Yaskawa INFORM job: KRIS4(-224_-90)X2.JBI

/JOB
//NAME KRIS4(-224_-90)X2
//POS
///NPOS 317,317,317,14,0,0
///TOOL 0
///POSTYPE PULSE
///PULSE
C00000=126,-73357,-105376,-18827,72039,-77556
C00001=32651,40852,-26417,-15259,84054,10521
C00002=30282,121459,21655,-7232,82256,-84550
C00003=119678,189491,121384,-6609,55844,-83781
C00004=119958,189291,121101,-6814,55937,-83682
C00005=119958,189291,121101,-6814,104918,-83682
C00006=69507,150313,105301,-6814,83622,-83682
C00007=102374,11647,-10601,-6208,113224,-88139
C00008=49110,-96581,-90191,-6208,113224,-88139
C00009=-73090,-118428,-105692,-6208,113224,-88139
C00010=-121621,-118428,-105692,-6208,113224,-88139
C00011=72199,118597,79738,-6814,89727,-83682
C00012=-14837,117754,79738,-6814,55937,-83682
C00013=-44504,100666,44561,-7265,69044,-83737
C00014=-106120,216,-72664,-1265,72875,-87293
C00015=-133015,-103640,-65816,3996,83698,-82063
C00016=-132086,-97485,-64003,4135,58701,-800
C00017=-149065,-104779,-51399,-7594,43822,-5087
C00018=-150289,-91952,-48932,-6393,56924,-6348
C00019=-150393,-90903,-46944,-6418,56235,-6345
C00020=-150312,-91064,-47459,-6419,56476,-6331
C00021=-149346,-88536,-46306,-6590,57139,-6001
C00022=-150281,-91600,-48374,-6405,56765,-6336
C00023=-170298,-72142,-39060,-11518,57888,-13007
C00024=-170167,-71928,-38964,-11546,57956,-12963
C00025=-170167,-71173,-37488,-11610,57441,-12905
C00026=-170167,-71393,-37919,-11591,57591,-12921
C00027=-169145,-69698,-37147,-11804,58123,-12578
C00028=-170288,-72356,-39514,-11498,58052,-13018
C00029=-137447,-116054,-63762,-19682,56909,112
C00030=-108026,-108792,-54867,4103,57296,6110
C00031=-81416,-94598,-46445,196,58741,15925
C00032=-81757,-93684,-45677,246,58738,15800
C00033=-81757,-92858,-44382,247,58365,15799
C00034=-81757,-93619,-45575,246,58708,15800
C00035=-82768,-91970,-45027,393,59221,15429
C00036=-81930,-94457,-46518,272,58858,15736
C00037=-128580,-105651,-52299,6719,58617,-1362
C00038=-130033,-102824,-49114,6921,58227,-1914
C00039=-130033,-101283,-46878,6964,57648,-1951
C00040=-130033,-101721,-47515,6952,57813,-1940
C00041=-129738,-99854,-46987,6872,58421,-1793
C00042=-130056,-102692,-48758,6935,58079,-1930
C00043=-106734,-120076,-67764,3834,59373,6657
C00044=-106734,-120076,-67764,3834,76101,81400
C00045=-85493,-101158,-51309,10056,72841,87538
C00046=-85426,-99920,-49312,10091,72250,87511
C00047=-85426,-98477,-47146,10119,71667,87460
C00048=-85426,-98764,-47576,10113,71783,87469
C00049=-84550,-100156,-47986,10204,71224,87714
C00050=-85920,-99324,-49419,10033,72673,87380
C00051=-152431,-100504,-49770,2471,77391,65939
C00052=-152805,-100536,-48996,2423,76908,65809
C00053=-152805,-99353,-47240,2427,76436,65801
C00054=-152805,-99697,-47754,2425,76574,65803
C00055=-153892,-101565,-48290,2277,75972,65442
C00056=-152767,-100966,-49728,2425,77135,65826
C00057=-175766,-86349,-42944,-18121,68088,61743
C00058=-175951,-86348,-42668,-18137,67889,61707
C00059=-175951,-85124,-40623,-18213,67291,61803
C00060=-175951,-85392,-41070,-18196,67421,61782
C00061=-177474,-87024,-41664,-18224,66648,61355
C00062=-175558,-86298,-43164,-18103,68288,61786
C00063=-175558,-91829,-52585,-17786,71106,61349
C00064=-197698,-109667,-58160,-17366,61060,54816
C00065=-219000,-104945,-43712,-24315,53908,49637
C00066=-231055,-104193,-38505,-23952,48237,46148
C00067=-233659,-103437,-37306,-23712,47268,45306
C00068=-233659,-102004,-35373,-23879,46852,45418
C00069=-233659,-102412,-35924,-23830,46971,45386
C00070=-237043,-102549,-35954,-23321,46092,44173
C00071=-233629,-103481,-37368,-23709,47288,45313
C00072=-215461,-127400,-43893,-16870,58722,48272
C00073=-218544,-127186,-42626,-17459,57581,47480
C00074=-218544,-125569,-40789,-17514,57295,47527
C00075=-220330,-126171,-41362,-17770,57042,47002
C00076=-227145,-126469,-41362,-18757,55731,45038
C00077=-215464,-127169,-42828,-16963,58209,48354
C00078=-177088,-126078,-40365,-8704,67148,58850
C00079=-153631,-128510,-40310,-2158,67069,65285
C00080=-133342,-128267,-39542,4651,67425,70358
C00081=-133342,-124673,-35501,4672,66785,70333
C00082=-133342,-124996,-35867,4671,66843,70335
C00083=-136291,-126982,-35925,3818,65972,69519
C00084=-133342,-126415,-37468,4662,67098,70344
C00085=-196611,-116316,-69487,-12664,87450,51098
C00086=-193209,-126845,-128640,-12422,104242,50582
C00087=-154889,-136514,-128640,-12422,104242,50582
C00088=49700,-188138,-128640,-12422,104242,50582
C00089=95044,-166675,-127403,-9604,101606,54242
C00090=100905,-121879,-41170,-2953,61354,-13811
C00091=47156,-125376,-41742,-10980,55894,-30486
C00092=47156,-123817,-39951,-11019,55598,-30455
C00093=47156,-124234,-40431,-11009,55677,-30464
C00094=51773,-123508,-40415,-10441,56507,-29089
C00095=47156,-124816,-41100,-10994,55787,-30475
C00096=106085,-127336,-41103,-2720,58495,-12699
C00097=106085,-127336,-41103,-2720,58495,-12699
C00098=106085,-125446,-38966,-2726,58152,-12693
C00099=106085,-125807,-39375,-2725,58219,-12694
C00100=107264,-124702,-39383,-2517,58821,-12358
C00101=106085,-127485,-41271,-2717,58524,-12702
C00102=100408,-120926,-37847,15529,71533,-19798
C00103=97019,-119074,-33059,14623,70083,-20929
C00104=97019,-117387,-31072,14654,69737,-20973
C00105=97019,-117741,-31491,14648,69810,-20964
C00106=98849,-116641,-31480,15187,70099,-20422
C00107=96336,-121085,-34976,14390,70314,-21090
C00108=117002,-126078,-36297,14353,59540,-14518
C00109=129547,-123648,-35340,18268,59922,-11292
C00110=117730,-128646,-41030,15406,62632,-14363
C00111=118409,-131302,-43968,5246,61629,-11067
C00112=120969,-131398,-38796,6988,54321,-10972
C00113=120206,-131306,-38746,6863,54384,-11194
C00114=120401,-140874,-53529,6577,58526,-10873
C00115=92949,-132183,-43651,2261,56631,-10244
C00116=85861,-128380,-38765,-239,57883,-11923
C00117=85623,-128366,-38766,-283,57890,-11992
C00118=82836,-128240,-39082,-8880,55261,-11515
C00119=99554,-124935,-41395,-6066,59525,-6766
C00120=106086,-187684,-135216,-4534,68260,-4839
C00121=27739,-169745,-128413,-4049,68845,15832
C00122=-73947,-156826,-135344,-2505,79379,12508
C00123=-156474,-127565,-44757,-2910,70220,64434
C00124=-184477,-125463,-34959,-7013,67471,54171
C00125=-136126,-128460,-34213,11142,64994,67622
C00126=-154263,-130476,-42112,2655,69883,62096
C00127=-171605,-138664,-45039,-640,62750,56909
C00128=-183285,-124480,-40863,-3523,67329,53581
C00129=-201708,-124095,-40052,-8196,65992,48445
C00130=-164693,-130393,-40095,1325,64018,58749
C00131=-142889,-132361,-46546,6897,66121,64856
C00132=-228263,-110324,-43358,-23728,50162,46686
C00133=-235581,-106051,-39851,-22875,48410,44119
C00134=-236443,-96869,-37709,-21687,51363,43058
C00135=-226552,-115005,-54629,-22549,54767,46269
C00136=-203481,-118873,-57487,-18716,57337,53342
C00137=-209230,-112060,-51294,-18356,55868,51433
C00138=-214685,-102612,-48820,-17221,57967,49003
C00139=-205976,-112243,-55103,-18172,58669,52173
C00140=-201958,-123065,-58725,-3253,73839,54936
C00141=-198681,-127844,-56028,-6414,64844,57079
C00142=-178104,-136485,-56885,-3962,62059,63635
C00143=-171824,-140203,-61595,-3068,63271,65534
C00144=-141766,-147898,-61645,3344,56480,74079
C00145=-136469,-141007,-56961,2843,60494,76114
C00146=-120497,-136999,-55124,10696,63094,79702
C00147=-164064,-147455,-64185,5609,61717,65893
C00148=-164064,-147455,-64185,5609,61717,65893
C00149=-130860,-150279,-64151,-6173,30547,-11978
C00150=-181055,-130986,-61566,17152,51608,-35195
C00151=-181843,-125511,-58523,17019,52654,-35316
C00152=-83956,-132387,-59007,-5944,41709,3692
C00153=-101244,-134284,-58376,7865,38480,-5637
C00154=-129711,-151516,-73375,17379,42716,-18129
C00155=-134581,-137990,-74595,-25751,56070,1389
C00156=-110654,-139179,-74777,-26363,62443,9081
C00157=-115870,-127626,-66583,-26250,61756,7273
C00158=-184118,-104582,-60976,-13857,52675,-18268
C00159=-171621,-128341,-75090,-18129,51623,-12881
C00160=-119711,-181360,-121572,-24950,66300,4723
C00161=-89347,-163256,-129350,-23289,87878,11502
C00162=-119711,-181360,-135603,-24950,39029,4723
C00163=-119711,-181360,-135603,-24950,39029,4723
C00164=-67118,-136665,-130676,-31892,63753,-5674
C00165=-40548,-161800,-132385,-30407,51173,2851
C00166=-38594,-160347,-135413,-37506,33521,-5777
C00167=-38158,-160025,-136084,-39080,61805,-7690
C00168=-9060,-155984,-136090,-36075,61852,-27249
C00169=-9060,-155984,-136090,-36075,61852,-27249
C00170=35778,-73357,-105376,-18827,72039,-77556
C00171=35778,-73357,-105376,-18827,72039,-77556
C00172=121972,-60692,-66036,-23906,48760,-72917
C00173=121972,-63565,-66036,-13351,77444,-72917
C00174=114761,-44204,-50669,-11461,76826,-75375
C00175=114807,-42889,-47501,-11529,75582,-75243
C00176=114807,-42796,-46589,-11554,75077,-75195
C00177=114807,-42822,-46844,-11546,75217,-75208
C00178=114733,-44587,-47920,-11539,74967,-75210
C00179=114807,-42889,-47501,-11529,75582,-75243
C00180=106693,-40989,-47922,8584,79047,-76853
C00181=106712,-40732,-46990,8589,78608,-76878
C00182=106712,-40651,-45975,8604,78031,-76918
C00183=106712,-40674,-46241,8599,78181,-76908
C00184=106551,-42339,-47274,8643,77981,-76977
C00185=106693,-40989,-47922,8584,79047,-76853
C00186=119731,-42339,-42353,28777,73600,-71789
C00187=120080,-41537,-40336,28806,72749,-71870
C00188=120080,-41293,-39100,28897,72189,-72014
C00189=120080,-41335,-39305,28882,72281,-71990
C00190=120073,-43216,-40463,28920,72059,-72050
C00191=120080,-41537,-40336,28806,72749,-71870
C00192=101589,-42073,-44271,32201,81327,-76893
C00193=104782,-94542,-85411,8339,74693,-77861
C00194=98731,-154827,-131308,9878,72678,-80158
C00195=98731,-154827,-131308,9878,72678,-80158
C00196=98731,-154827,-131308,9878,72678,-80158
C00197=141095,-137804,-121947,-4358,90462,-65341
C00198=171917,-153174,-112370,11397,78411,-54227
C00199=199110,-110397,-63847,11158,69278,-59316
C00200=199661,-105459,-60576,13729,71348,-59282
C00201=199661,-104714,-59434,13753,71034,-59321
C00202=199661,-104881,-59692,13747,71104,-59313
C00203=201697,-105978,-60019,13785,70422,-58683
C00204=199661,-105459,-60576,13729,71348,-59282
C00205=123960,-138876,-68675,7989,69585,-84604
C00206=124072,-138705,-67366,8043,68864,-84619
C00207=124072,-137612,-66165,8049,68688,-84634
C00208=124072,-137824,-66399,8047,68723,-84632
C00209=124282,-139731,-66590,8126,67850,-84627
C00210=124072,-138655,-67314,8040,68857,-84622
C00211=114984,-139242,-68510,-12959,69151,-83072
C00212=114827,-138670,-67011,-13034,68516,-83052
C00213=114827,-136931,-65095,-13059,68238,-83020
C00214=114827,-137199,-65392,-13055,68282,-83025
C00215=114467,-139013,-65570,-13183,67430,-83044
C00216=114827,-138670,-67011,-13034,68516,-83052
C00217=133085,-142772,-85485,-9589,79895,-78262
C00218=119908,-107051,-70579,-11526,87272,-83253
C00219=119905,-107270,-70562,-11527,87152,-83243
C00220=119905,-106417,-69135,-11528,86722,-83203
C00221=119905,-106577,-69401,-11528,86804,-83211
C00222=119887,-108279,-69933,-11533,86265,-83166
C00223=119905,-107341,-70681,-11527,87191,-83247
C00224=147950,-101609,-70952,8097,88078,-75282
C00225=148936,-101577,-69519,8210,87121,-75014
C00226=148936,-100979,-68423,8210,86757,-75037
C00227=148936,-101159,-68752,8210,86867,-75032
C00228=149395,-102566,-69230,8263,86398,-74908
C00229=148936,-101830,-69986,8210,87277,-75005
C00230=165354,-89650,-65481,16319,85072,-70011
C00231=165779,-89873,-64407,16347,84242,-69973
C00232=165779,-89214,-62991,16359,83730,-70041
C00233=165779,-89312,-63202,16357,83805,-70031
C00234=166355,-90439,-63644,16386,83393,-69883
C00235=165632,-89756,-64683,16338,84492,-69992
C00236=143601,-106428,-78314,14904,88558,-77172
C00237=127839,-150907,-89343,18520,59767,-2936
C00238=132953,-138286,-79588,18019,59168,-1112
C00239=137115,-133470,-77672,17386,59565,529
C00240=137115,-131953,-75830,17447,59223,475
C00241=137115,-132842,-76915,17411,59423,507
C00242=136304,-129881,-76308,17304,60683,404
C00243=137115,-133253,-77414,17394,59515,521
C00244=181699,-110020,-71549,8619,60587,17610
C00245=181630,-109868,-71398,8637,60579,17583
C00246=181630,-109061,-70095,8670,60195,17555
C00247=181630,-109567,-70911,8650,60436,17574
C00248=179495,-107200,-70173,9064,61418,16842
C00249=181374,-109783,-71626,8682,60786,17501
C00250=138549,-156108,-92608,17680,56945,638
C00251=92857,-152389,-93170,-1138,51221,-11865
C00252=89241,-137374,-84375,-135,53495,-13313
C00253=89241,-137236,-84209,-135,53464,-13313
C00254=89241,-136248,-83020,-135,53240,-13313
C00255=89241,-136629,-83479,-135,53327,-13313
C00256=90422,-134246,-82978,-442,54247,-12852
C00257=88987,-137859,-84464,-69,53301,-13413
C00258=151501,-140988,-86034,-14129,58291,10466
C00259=150678,-138310,-84494,-13941,58574,10114
C00260=150678,-137164,-83136,-13977,58332,10146
C00261=150678,-137515,-83554,-13966,58407,10136
C00262=149186,-134345,-82896,-13563,59357,9449
C00263=151128,-139683,-85226,-14047,58399,10308
C00264=153806,-132474,-82078,-14195,60563,11039
C00265=88294,-133814,-82651,111,54267,-13684
C00266=119170,-146244,-89248,-14851,56054,5885
C00267=129919,-160370,-92966,12704,53201,-3154
C00268=134642,-143084,-81504,11683,54346,-1201
C00269=167270,-136117,-75530,1628,46891,11778
C00270=184998,-113755,-66262,10763,44700,16651
C00271=164928,-143381,-78407,9170,42235,9240
C00272=155273,-152427,-83467,13136,41921,4825
C00273=158141,-110882,-79211,11782,79402,-69500
C00274=156021,-110302,-75029,11867,77473,-70419
C00275=165528,-106206,-70771,11800,75600,-67301
C00276=175934,-96636,-67342,11366,76879,-63551
C00277=131080,-121620,-80305,3109,79327,-78003
C00278=138412,-119763,-75738,-25,77941,-75181
C00279=121865,-121897,-76297,-1096,77077,-80681
C00280=118816,-123903,-80121,-1281,78355,-81709
C00281=109990,-123163,-79929,-1817,78452,-84652
C00282=123486,-121654,-75594,-8156,77182,-79251
C00283=148715,-110583,-64793,-26650,87105,-69201
C00284=135969,-121502,-76764,-18008,81762,-74135
C00285=154667,-142334,-81197,-15526,77761,-67286
C00286=153773,-135579,-66423,-14508,74760,-67487
C00287=169136,-136018,-63121,-11093,74659,-62747
C00288=139166,-140952,-63595,-17941,67950,-71134
C00289=148278,-138995,-66659,-15795,72315,-68901
C00290=144415,-140880,-69264,8833,65243,-74412
C00291=148924,-141501,-67458,9395,63396,-73104
C00292=174434,-134936,-66673,11173,63406,-64720
C00293=167439,-135845,-70174,10586,65898,-66819
C00294=192902,-115042,-63146,20265,60680,-60371
C00295=201183,-110866,-58973,19481,58401,-57610
C00296=207998,-99743,-55745,17878,60466,-54609
C00297=170801,-131743,-76226,21430,65470,-67743
C00298=164740,-137810,-91614,20635,72894,-68588
C00299=164740,-137810,-91614,20635,72894,-68588
C00300=149447,-191890,-120181,21381,67024,-75156
C00301=149584,-192173,-120256,21405,66899,-75131
C00302=149584,-192173,-120256,21405,66899,-75131
C00303=114761,-44204,-50669,-11461,76826,-75375
C00304=117531,-39747,-45231,-12087,78952,-74614
C00305=125622,-38648,-38317,-31754,77240,-72218
C00306=114060,-50823,-52718,-11111,71580,-75110
C00307=124826,-51246,-53710,3634,72889,-70409
C00308=127047,-37417,-44991,3423,81297,-69380
C00309=134341,-35671,-43811,1894,81230,-66916
C00310=133954,-36259,-45628,1970,82055,-67034
C00311=135284,-28260,-32637,27547,76219,-65313
C00312=136540,-27437,-30649,27351,75093,-65095
C00313=137370,-25955,-24515,36210,70473,-65832
C00314=131832,-52683,-49405,33204,65462,-69826
C00315=109380,-75662,-60137,33198,63885,-64520
C00316=9054,-143647,-113334,-5954,77551,-79151
BC00000=192636,515545,1075136
BC00001=106856,514699,1075147
BC00002=45026,513209,1075136
BC00003=297205,515545,1075136
BC00004=388258,132939,1075136
BC00005=388258,132939,1075136
BC00006=266781,91691,1075136
BC00007=338196,12076,1075135
BC00008=385019,2960,1075135
BC00009=385019,2960,1075135
BC00010=335835,2960,1075135
BC00011=245343,24956,1075136
BC00012=171885,-116810,981693
BC00013=145068,-168564,1075136
BC00014=282408,-168564,1075136
BC00015=324871,12764,1075136
BC00016=324871,12764,1033476
BC00017=324871,12764,1033476
BC00018=324871,12764,1033476
BC00019=324871,12764,1033476
BC00020=324871,12764,1033476
BC00021=324871,12764,1033476
BC00022=324871,12764,1033476
BC00023=324871,12764,1033476
BC00024=324871,12764,1033476
BC00025=324871,12764,1033476
BC00026=324871,12764,1033476
BC00027=324871,12764,1033476
BC00028=324871,12764,1033476
BC00029=324871,12764,1033476
BC00030=324871,12764,1033476
BC00031=324871,12764,1033476
BC00032=324871,12764,1033476
BC00033=324871,12764,1033476
BC00034=324871,12764,1033476
BC00035=324871,12764,1033476
BC00036=324871,12764,1033476
BC00037=324871,12764,1033476
BC00038=324871,12764,1033476
BC00039=324871,12764,1033476
BC00040=324871,12764,1033476
BC00041=324871,12764,1033476
BC00042=324871,12764,1033476
BC00043=324871,12764,1033476
BC00044=324871,42664,1033476
BC00045=324871,42664,1033476
BC00046=324871,42664,1033476
BC00047=324871,42664,1033476
BC00048=324871,42664,1033476
BC00049=324871,42664,1033476
BC00050=324871,42664,1033476
BC00051=324871,42664,1033476
BC00052=324871,42664,1033476
BC00053=324871,42664,1033476
BC00054=324871,42664,1033476
BC00055=324871,42664,1033476
BC00056=324871,42664,1033476
BC00057=324871,42664,1033476
BC00058=324871,42664,1033476
BC00059=324871,42664,1033476
BC00060=324871,42664,1033476
BC00061=324871,42664,1033476
BC00062=324871,42664,1033476
BC00063=324871,42664,1033476
BC00064=324871,42664,1033476
BC00065=324871,70402,1033476
BC00066=324871,70402,1033476
BC00067=324871,70402,1033476
BC00068=324871,70402,1033476
BC00069=324871,70402,1033476
BC00070=324871,70402,1033476
BC00071=324871,70402,1033476
BC00072=324871,70402,1033476
BC00073=324871,70402,1033476
BC00074=324871,70402,1033476
BC00075=324871,70402,1033476
BC00076=324871,70402,1033476
BC00077=324871,70402,1033476
BC00078=346902,67759,1033476
BC00079=365604,67759,1033476
BC00080=358835,67759,1033476
BC00081=358835,67759,1033476
BC00082=358835,67759,1033476
BC00083=358835,67759,1033476
BC00084=358835,67759,1033476
BC00085=338593,67759,1033476
BC00086=365604,66159,1034603
BC00087=365604,17709,1034603
BC00088=365604,1629,1034603
BC00089=299593,3037,1034603
BC00090=314294,3037,1034603
BC00091=350319,4086,1007387
BC00092=350319,4086,1007387
BC00093=350319,4086,1007387
BC00094=350319,4086,1007387
BC00095=350319,4086,1007387
BC00096=302029,3926,1031408
BC00097=301345,10358,1012837
BC00098=301345,10358,1012837
BC00099=301345,10358,1012837
BC00100=301345,10358,1012837
BC00101=301345,10358,1012837
BC00102=302371,1302,1012837
BC00103=302371,1302,1012837
BC00104=302371,1302,1012837
BC00105=302371,1302,1012837
BC00106=302371,1302,1012837
BC00107=302371,1302,1012837
BC00108=302371,1302,1012837
BC00109=292881,1302,1012837
BC00110=310946,1302,1012837
BC00111=309160,1302,1012837
BC00112=309160,1302,1012837
BC00113=322422,1302,1012837
BC00114=322422,1302,1012837
BC00115=365717,2550,1012837
BC00116=365717,2550,1012837
BC00117=365717,2550,1012837
BC00118=365717,2550,1012837
BC00119=344627,2742,1042919
BC00120=344627,2742,1042919
BC00121=350887,22143,1073092
BC00122=276696,2854,1073092
BC00123=365604,67759,1033476
BC00124=354680,71198,1033476
BC00125=354680,71198,1033476
BC00126=354680,71198,1033476
BC00127=289396,71198,1033476
BC00128=299083,59780,1033476
BC00129=299083,59780,1033476
BC00130=299083,59780,1033476
BC00131=299083,59780,1033476
BC00132=323021,69640,1018791
BC00133=323021,69640,1018791
BC00134=323021,69640,1018791
BC00135=323021,69640,1018791
BC00136=323021,86344,1018791
BC00137=323020,86342,1018791
BC00138=323021,86344,1018791
BC00139=323021,86344,1018791
BC00140=323021,86344,1018791
BC00141=323021,86344,1018791
BC00142=323021,86344,1018791
BC00143=323021,86344,1018791
BC00144=359311,86344,1018791
BC00145=359311,86344,1018791
BC00146=359311,86344,1018791
BC00147=359311,86344,1018791
BC00148=320650,86344,1061699
BC00149=320650,38724,1061699
BC00150=348099,38724,988490
BC00151=348099,38724,988490
BC00152=348099,38724,988490
BC00153=348097,38726,988489
BC00154=348099,38724,988490
BC00155=348099,38724,988490
BC00156=317547,52292,963745
BC00157=317547,52292,963745
BC00158=317547,52292,963745
BC00159=317547,52292,963745
BC00160=317547,31600,963745
BC00161=278487,3584,1056780
BC00162=340345,-44387,1068891
BC00163=340345,-123490,1068891
BC00164=331767,-1766,1070081
BC00165=234698,5049,1063085
BC00166=254493,47555,1069374
BC00167=326806,106778,1070769
BC00168=344384,299723,1072198
BC00169=344384,446401,1072198
BC00170=295310,515545,1075136
BC00171=295310,513516,1075136
BC00172=295310,513263,813287
BC00173=335993,429318,731212
BC00174=335993,429318,731212
BC00175=335993,429318,731212
BC00176=335993,429318,731212
BC00177=335993,429318,731212
BC00178=335993,429318,731212
BC00179=335993,429318,731212
BC00180=292293,429318,731212
BC00181=292293,429318,731212
BC00182=292293,429318,731212
BC00183=292293,429318,731212
BC00184=292293,429318,731212
BC00185=292293,429318,731212
BC00186=292293,429318,731212
BC00187=292293,429318,731212
BC00188=292293,429318,731212
BC00189=292293,429318,731212
BC00190=292293,429318,731212
BC00191=292293,429318,731212
BC00192=292293,429318,731212
BC00193=292293,429318,731212
BC00194=292293,429318,979834
BC00195=314373,292172,979834
BC00196=314373,275872,695664
BC00197=349600,266255,695664
BC00198=349600,243768,695664
BC00199=318481,229664,891298
BC00200=318481,229664,891298
BC00201=318481,229664,891298
BC00202=318481,229664,891298
BC00203=318481,229664,891298
BC00204=318481,229664,891298
BC00205=318481,229664,891298
BC00206=318481,229664,891298
BC00207=318481,229664,891298
BC00208=318481,229664,891298
BC00209=318481,229664,891298
BC00210=318481,229664,891298
BC00211=347990,229664,891297
BC00212=347990,229664,891297
BC00213=347990,229664,891297
BC00214=347990,229664,891297
BC00215=347990,229664,891297
BC00216=347990,229664,891297
BC00217=347990,229664,891297
BC00218=347990,229664,891297
BC00219=347990,229664,891297
BC00220=347990,229664,891297
BC00221=347990,229664,891297
BC00222=347990,229664,891297
BC00223=347990,229664,891297
BC00224=347990,229664,891297
BC00225=347990,229664,891297
BC00226=347990,229664,891297
BC00227=347990,229664,891297
BC00228=347990,229664,891297
BC00229=347990,229664,891297
BC00230=317379,229664,891297
BC00231=317379,229664,891297
BC00232=317379,229664,891297
BC00233=317379,229664,891297
BC00234=317379,229664,891297
BC00235=317379,229664,891297
BC00236=317379,229664,891297
BC00237=317379,229664,891297
BC00238=317379,229664,891297
BC00239=317379,229664,891297
BC00240=317379,229664,891297
BC00241=317379,229664,891297
BC00242=317379,229664,891297
BC00243=317379,229664,891297
BC00244=317379,229664,891297
BC00245=317379,229664,891297
BC00246=317379,229664,891297
BC00247=317379,229664,891297
BC00248=317379,229664,891297
BC00249=317379,229664,891297
BC00250=317379,229664,891297
BC00251=339726,229664,891297
BC00252=339725,229663,891294
BC00253=339725,229663,891294
BC00254=339725,229663,891294
BC00255=339725,229663,891294
BC00256=339725,229663,891294
BC00257=339725,229663,891294
BC00258=339725,229663,891294
BC00259=339725,229663,891294
BC00260=339725,229663,891294
BC00261=339725,229663,891294
BC00262=339725,229663,891294
BC00263=339725,229663,891294
BC00264=339725,229663,891294
BC00265=339725,229663,891294
BC00266=339725,229663,891294
BC00267=310311,229663,891294
BC00268=310311,229663,891294
BC00269=310311,229663,891294
BC00270=310311,229663,891294
BC00271=310311,229663,891294
BC00272=310311,229663,891294
BC00273=310311,229663,891294
BC00274=310311,229663,891294
BC00275=310311,229663,891294
BC00276=310311,229663,891294
BC00277=310311,229663,891294
BC00278=310311,229663,891294
BC00279=310311,229663,891290
BC00280=310311,229663,891290
BC00281=351185,229663,891290
BC00282=351185,229663,891290
BC00283=351184,229663,891289
BC00284=351185,229663,891290
BC00285=351185,229663,891290
BC00286=351185,229663,891290
BC00287=351185,229663,891290
BC00288=351185,229663,891290
BC00289=351185,229663,891290
BC00290=335351,229663,891290
BC00291=335351,229663,891290
BC00292=335351,229663,891290
BC00293=335351,229663,891290
BC00294=335351,229663,891290
BC00295=335351,229663,891290
BC00296=335351,229663,891290
BC00297=335351,229663,891290
BC00298=335351,229663,891290
BC00299=352732,229663,1069777
BC00300=352732,229663,1069777
BC00301=352732,347909,1069777
BC00302=352732,347909,743295
BC00303=335993,429318,731212
BC00304=335994,429318,731211
BC00305=335994,429317,731208
BC00306=335994,429318,731211
BC00307=335994,429318,731211
BC00308=335994,429318,731211
BC00309=335994,429318,731211
BC00310=335994,429318,731211
BC00311=335994,429318,731211
BC00312=335994,429318,731211
BC00313=335994,429318,731211
BC00314=335994,429318,731211
BC00315=361465,487090,979283
BC00316=361465,516139,979283
EC00000=1986524,372644
EC00001=1986524,372644
EC00002=1986524,372644
EC00003=1986524,372644
EC00004=1986524,372644
EC00005=1986524,372644
EC00006=1986524,372644
EC00007=1986527,372644
EC00008=1986527,372644
EC00009=1986527,372644
EC00010=1986527,372644
EC00011=1986524,372644
EC00012=1986524,372644
EC00013=1986524,372644
EC00014=1986524,372644
EC00015=1986524,372644
EC00016=1986524,372644
EC00017=1986524,372644
EC00018=1986524,372644
EC00019=1986524,372644
EC00020=1986524,372644
EC00021=1986524,372644
EC00022=1986524,372644
EC00023=1986524,372644
EC00024=1986524,372644
EC00025=1986524,372644
EC00026=1986524,372644
EC00027=1986524,372644
EC00028=1986524,372644
EC00029=1986524,372644
EC00030=1986524,372644
EC00031=1986524,372644
EC00032=1986524,372644
EC00033=1986524,372644
EC00034=1986524,372644
EC00035=1986524,372644
EC00036=1986524,372644
EC00037=1986524,372644
EC00038=1986524,372644
EC00039=1986524,372644
EC00040=1986524,372644
EC00041=1986524,372644
EC00042=1986524,372644
EC00043=1986524,372644
EC00044=1986524,372644
EC00045=1986524,372644
EC00046=1986524,372644
EC00047=1986524,372644
EC00048=1986524,372644
EC00049=1986524,372644
EC00050=1986524,372644
EC00051=1986524,372644
EC00052=1986524,372644
EC00053=1986524,372644
EC00054=1986524,372644
EC00055=1986524,372644
EC00056=1986524,372644
EC00057=1986524,372644
EC00058=1986524,372644
EC00059=1986524,372644
EC00060=1986524,372644
EC00061=1986524,372644
EC00062=1986524,372644
EC00063=1986524,372644
EC00064=1986524,372644
EC00065=1986524,372644
EC00066=1986524,372644
EC00067=1986524,372644
EC00068=1986524,372644
EC00069=1986524,372644
EC00070=1986524,372644
EC00071=1986524,372644
EC00072=1986524,372644
EC00073=1986524,372644
EC00074=1986524,372644
EC00075=1986524,372644
EC00076=1986524,372644
EC00077=1986524,372644
EC00078=1986524,372644
EC00079=1986524,372644
EC00080=1986524,372644
EC00081=1986524,372644
EC00082=1986524,372644
EC00083=1986524,372644
EC00084=1986524,372644
EC00085=1986524,372644
EC00086=1986524,372644
EC00087=1986524,372644
EC00088=1986524,372644
EC00089=1986524,372644
EC00090=1986524,372644
EC00091=1986524,372644
EC00092=1986524,372644
EC00093=1986524,372644
EC00094=1986524,372644
EC00095=1986524,372644
EC00096=1986524,372644
EC00097=1986524,372644
EC00098=1986524,372644
EC00099=1986524,372644
EC00100=1986524,372644
EC00101=1986524,372644
EC00102=1986524,372644
EC00103=1986524,372644
EC00104=1986524,372644
EC00105=1986524,372644
EC00106=1986524,372644
EC00107=1986524,372644
EC00108=1986524,372644
EC00109=1986524,372644
EC00110=1986524,372644
EC00111=1986524,372644
EC00112=1986524,372644
EC00113=1986524,372644
EC00114=1986524,372644
EC00115=1986524,372644
EC00116=1986524,372644
EC00117=1986524,372644
EC00118=1986524,372644
EC00119=1986524,372644
EC00120=1986524,372644
EC00121=1986524,372644
EC00122=1986524,372644
EC00123=1986524,372644
EC00124=1986524,372644
EC00125=1986524,372644
EC00126=1986524,372644
EC00127=1986524,372644
EC00128=1986524,372644
EC00129=1986524,372644
EC00130=1986524,372644
EC00131=1986524,372644
EC00132=1986524,372644
EC00133=1986524,372644
EC00134=1986524,372644
EC00135=1986524,372644
EC00136=1986524,372644
EC00137=1986526,372644
EC00138=1986524,372644
EC00139=1986524,372644
EC00140=1986524,372644
EC00141=1986524,372644
EC00142=1986524,372644
EC00143=1986524,372644
EC00144=1986524,372644
EC00145=1986524,372644
EC00146=1986524,372644
EC00147=1986524,372644
EC00148=1986524,372644
EC00149=1986524,372644
EC00150=1986524,372644
EC00151=1986524,372644
EC00152=1986524,372644
EC00153=1986527,372644
EC00154=1986524,372644
EC00155=1986524,372644
EC00156=1986524,372644
EC00157=1986524,372644
EC00158=1986524,372644
EC00159=1986524,372644
EC00160=1986524,372644
EC00161=1986524,372644
EC00162=1986524,372644
EC00163=1986524,372644
EC00164=1924386,269829
EC00165=1942317,299498
EC00166=1898227,226544
EC00167=1888448,210364
EC00168=1813786,86826
EC00169=1813786,86826
EC00170=1660311,-167120
EC00171=1178646,-738387
EC00172=1144025,-740308
EC00173=1144025,-740308
EC00174=1144025,-740308
EC00175=1144025,-740308
EC00176=1144025,-740308
EC00177=1144025,-740308
EC00178=1144025,-740308
EC00179=1144025,-740308
EC00180=1144025,-740308
EC00181=1144025,-740308
EC00182=1144025,-740308
EC00183=1144025,-740308
EC00184=1144025,-740308
EC00185=1144025,-740308
EC00186=1144025,-740308
EC00187=1144025,-740308
EC00188=1144025,-740308
EC00189=1144025,-740308
EC00190=1144025,-740308
EC00191=1144025,-740308
EC00192=1144025,-740308
EC00193=1144025,-740308
EC00194=1144025,-740308
EC00195=1144025,-740308
EC00196=1144025,-740308
EC00197=1144025,-740308
EC00198=1144025,-740308
EC00199=1144025,-740308
EC00200=1144025,-740308
EC00201=1144025,-740308
EC00202=1144025,-740308
EC00203=1144025,-740308
EC00204=1144025,-740308
EC00205=1144025,-740308
EC00206=1144025,-740308
EC00207=1144025,-740308
EC00208=1144025,-740308
EC00209=1144025,-740308
EC00210=1144025,-740308
EC00211=1144023,-740308
EC00212=1144023,-740308
EC00213=1144023,-740308
EC00214=1144023,-740308
EC00215=1144023,-740308
EC00216=1144023,-740308
EC00217=1144023,-740308
EC00218=1144023,-740308
EC00219=1144023,-740308
EC00220=1144023,-740308
EC00221=1144023,-740308
EC00222=1144023,-740308
EC00223=1144023,-740308
EC00224=1144023,-740308
EC00225=1144023,-740308
EC00226=1144023,-740308
EC00227=1144023,-740308
EC00228=1144023,-740308
EC00229=1144023,-740308
EC00230=1144023,-740308
EC00231=1144023,-740308
EC00232=1144023,-740308
EC00233=1144023,-740308
EC00234=1144023,-740308
EC00235=1144023,-740308
EC00236=1144023,-740308
EC00237=1144023,-740308
EC00238=1144023,-740308
EC00239=1144023,-740308
EC00240=1144023,-740308
EC00241=1144023,-740308
EC00242=1144023,-740308
EC00243=1144023,-740308
EC00244=1144023,-740308
EC00245=1144023,-740308
EC00246=1144023,-740308
EC00247=1144023,-740308
EC00248=1144023,-740308
EC00249=1144023,-740308
EC00250=1144023,-740308
EC00251=1144023,-740308
EC00252=1144020,-740308
EC00253=1144020,-740308
EC00254=1144020,-740308
EC00255=1144020,-740308
EC00256=1144020,-740308
EC00257=1144020,-740308
EC00258=1144020,-740308
EC00259=1144020,-740308
EC00260=1144020,-740308
EC00261=1144020,-740308
EC00262=1144020,-740308
EC00263=1144020,-740308
EC00264=1144019,-740308
EC00265=1144019,-740308
EC00266=1144019,-740308
EC00267=1144019,-740308
EC00268=1144019,-740308
EC00269=1144019,-740308
EC00270=1144019,-740308
EC00271=1144019,-740308
EC00272=1144019,-740308
EC00273=1144019,-740308
EC00274=1144019,-740308
EC00275=1144019,-740308
EC00276=1144019,-740308
EC00277=1144019,-740308
EC00278=1144019,-740308
EC00279=1144018,-740308
EC00280=1144018,-740308
EC00281=1144018,-740308
EC00282=1144018,-740308
EC00283=1144017,-740308
EC00284=1144018,-740308
EC00285=1144018,-740308
EC00286=1144018,-740308
EC00287=1144018,-740308
EC00288=1144018,-740308
EC00289=1144018,-740308
EC00290=1144018,-740308
EC00291=1144018,-740308
EC00292=1144018,-740308
EC00293=1144018,-740308
EC00294=1144018,-740308
EC00295=1144018,-740308
EC00296=1144018,-740308
EC00297=1144018,-740308
EC00298=1144018,-740308
EC00299=1144018,-740308
EC00300=1144018,-740308
EC00301=1144018,-740308
EC00302=1144018,-740308
EC00303=1144025,-740308
EC00304=1144023,-740309
EC00305=1144020,-740309
EC00306=1144023,-740309
EC00307=1144023,-740309
EC00308=1144023,-740309
EC00309=1144023,-740309
EC00310=1144023,-740309
EC00311=1144023,-740309
EC00312=1144023,-740309
EC00313=1144023,-740309
EC00314=1144023,-740309
EC00315=1144023,-740309
EC00316=1207380,-740309
///POSTYPE BASE
///RECTAN
///RCONF 0,0,0,0,1,0,0,0,0,0,0,0,0,0,0,0,0,0,0,0,0,0,0,0
P00006=2.006,1.622,-0.565,0.0000,0.0000,0.0000
P00021=0.073,2.058,-0.109,0.0000,0.0000,0.0000
P00022=2.006,1.622,-0.565,0.0000,0.0000,0.0000
///RCONF 0,0,0,0,0,0,0,0,0,0,0,0,0,0,0,0,0,0,0,0,0,0,0,0
P00023=-2.957,-4.083,2.762,0.0000,0.0000,0.0000
P00024=-1.466,-0.226,-0.419,0.0000,0.0000,0.0000
P00025=3.643,0.007,-2.585,0.0000,0.0000,0.0000
P00026=2.644,0.055,-2.583,0.0000,0.0000,0.0000
P00027=2.278,0.099,-4.210,0.0000,0.0000,0.0000
P00028=-1.778,-0.182,-2.050,0.0000,0.0000,0.0000
P00029=1.749,4.006,-0.261,0.0000,0.0000,0.0000
P00030=-0.014,-0.768,0.131,0.0000,0.0000,0.0000
P00031=-0.170,0.039,-0.647,0.0000,0.0000,0.0000
P00032=-0.423,0.157,3.222,0.0000,0.0000,0.0000
P00033=0.854,-1.099,3.047,0.0000,0.0000,0.0000
//INST
///DATE 2024/12/09 22:39
///ATTR SC,RW
///GROUP1 RB1,BS1
///GROUP2 ST1
NOP
'300124 MUZYLO
MOVJ C00000 BC00000 VJ=100.00  +MOVJ EC00000 VJ=100.00
CALL JOB:CLEAN-R1_KM_NEW
MOVJ C00001 BC00001 VJ=100.00  +MOVJ EC00001 VJ=100.00
MOVJ C00002 BC00002 VJ=100.00  +MOVJ EC00002 VJ=100.00
MOVJ C00003 BC00003 VJ=100.00  +MOVJ EC00003 VJ=100.00
MOVJ C00004 BC00004 VJ=100.00  +MOVJ EC00004 VJ=100.00
MOVJ C00005 BC00005 VJ=100.00  +MOVJ EC00005 VJ=0.78
MOVJ C00006 BC00006 VJ=100.00  +MOVJ EC00006 VJ=100.00
MOVJ C00007 BC00007 VJ=60.00  +MOVJ EC00007 VJ=60.00
MOVJ C00008 BC00008 VJ=60.00  +MOVJ EC00008 VJ=60.00
MOVJ C00009 BC00009 VJ=60.00  +MOVJ EC00009 VJ=60.00
MOVJ C00010 BC00010 VJ=60.00  +MOVJ EC00010 VJ=60.00
COMM MOVJ C00011 BC00011 VJ=100.00  +MOVJ EC00011 VJ=100.00
COMM MOVJ C00012 BC00012 VJ=100.00  +MOVJ EC00012 VJ=100.00
COMM MOVJ C00013 BC00013 VJ=100.00  +MOVJ EC00013 VJ=100.00
COMM MOVJ C00014 BC00014 VJ=100.00  +MOVJ EC00014 VJ=100.00
COMM MOVJ C00015 BC00015 VJ=100.00  +MOVJ EC00015 VJ=100.00
COMM MOVJ C00016 BC00016 VJ=100.00  +MOVJ EC00016 VJ=100.00
MOVJ C00017 BC00017 VJ=100.00  +MOVJ EC00017 VJ=100.00
SMOVL C00018 BC00018 V=100.0  +MOVJ EC00018
SREFP 3 C00019 BC00019  +REFP EC00019
CALL JOB:SEARCH-R1-S13D
SET P032 P006
SFTON3D P032
SMOVL C00020 BC00020 V=100.0  +MOVJ EC00020
SREFP 3 C00021 BC00021  +REFP EC00021
CALL JOB:SEARCH-R1-S13D
SET P032 P006
SFTON3D P032
SMOVL C00022 BC00022 V=100.0  +MOVJ EC00022
SFTOF3D
SMOVL C00023 BC00023 V=333.3  +MOVJ EC00023
SMOVL C00024 BC00024 V=100.0  +MOVJ EC00024
SREFP 3 C00025 BC00025  +REFP EC00025
CALL JOB:SEARCH-R1-S13D
SET P033 P006
SFTON3D P033
SMOVL C00026 BC00026 V=100.0  +MOVJ EC00026
SREFP 3 C00027 BC00027  +REFP EC00027
CALL JOB:SEARCH-R1-S13D
SET P033 P006
SFTON3D P033
SMOVL C00028 BC00028 V=100.0  +MOVJ EC00028
SFTOF3D
SMOVL C00029 BC00029 V=333.3  +MOVJ EC00029
SMOVL C00030 BC00030 V=1000.0  +MOVJ EC00030
SMOVL C00031 BC00031 V=666.7  +MOVJ EC00031
SMOVL C00032 BC00032 V=100.0  +MOVJ EC00032
SREFP 3 C00033 BC00033  +REFP EC00033
CALL JOB:SEARCH-R1-S13D
SET P030 P006
SFTON3D P030
SMOVL C00034 BC00034 V=100.0  +MOVJ EC00034
SREFP 3 C00035 BC00035  +REFP EC00035
CALL JOB:SEARCH-R1-S13D
SET P030 P006
SFTON3D P030
SMOVL C00036 BC00036 V=100.0  +MOVJ EC00036
SFTOF3D
SMOVL C00037 BC00037 V=666.7  +MOVJ EC00037
SMOVL C00038 BC00038 V=100.0  +MOVJ EC00038
SREFP 3 C00039 BC00039  +REFP EC00039
CALL JOB:SEARCH-R1-S13D
SET P031 P006
SFTON3D P031
SMOVL C00040 BC00040 V=100.0  +MOVJ EC00040
SREFP 3 C00041 BC00041  +REFP EC00041
CALL JOB:SEARCH-R1-S13D
SET P031 P006
SFTON3D P031
SMOVL C00042 BC00042 V=100.0  +MOVJ EC00042
SFTOF3D
MOVJ C00043 BC00043 VJ=100.00  +MOVJ EC00043 VJ=100.00
MOVJ C00044 BC00044 VJ=100.00  +MOVJ EC00044 VJ=50.00
MOVJ C00045 BC00045 VJ=100.00  +MOVJ EC00045 VJ=50.00
SMOVL C00046 BC00046 V=100.0  +MOVJ EC00046
SREFP 3 C00047 BC00047  +REFP EC00047
CALL JOB:SEARCH-R1-S13D
SET P021 P006
SFTON3D P021
SMOVL C00048 BC00048 V=100.0  +MOVJ EC00048
SREFP 3 C00049 BC00049  +REFP EC00049
CALL JOB:SEARCH-R1-S13D
SET P021 P006
SFTON3D P021
SMOVL C00050 BC00050 V=100.0  +MOVJ EC00050
SFTOF3D
SMOVL C00051 BC00051 V=666.7  +MOVJ EC00051
SMOVL C00052 BC00052 V=100.0  +MOVJ EC00052
SREFP 3 C00053 BC00053  +REFP EC00053
CALL JOB:SEARCH-R1-S13D
SET P022 P006
SFTON3D P022
SMOVL C00054 BC00054 V=100.0  +MOVJ EC00054
SREFP 3 C00055 BC00055  +REFP EC00055
CALL JOB:SEARCH-R1-S13D
SET P022 P006
SFTON3D P022
SMOVL C00056 BC00056 V=100.0  +MOVJ EC00056
SFTOF3D
SMOVL C00057 BC00057 V=666.7  +MOVJ EC00057
SMOVL C00058 BC00058 V=100.0  +MOVJ EC00058
SREFP 3 C00059 BC00059  +REFP EC00059
CALL JOB:SEARCH-R1-S13D
SET P023 P006
SFTON3D P023
SMOVL C00060 BC00060 V=100.0  +MOVJ EC00060
SREFP 3 C00061 BC00061  +REFP EC00061
CALL JOB:SEARCH-R1-S13D
SET P023 P006
SFTON3D P023
SMOVL C00062 BC00062 V=100.0  +MOVJ EC00062
SFTOF3D
SMOVL C00063 BC00063 V=1000.0  +MOVJ EC00063
SMOVL C00064 BC00064 V=333.3  +MOVJ EC00064
SMOVL C00065 BC00065 V=333.3  +MOVJ EC00065
SMOVL C00066 BC00066 V=333.3  +MOVJ EC00066
SMOVL C00067 BC00067 V=100.0  +MOVJ EC00067
SREFP 3 C00068 BC00068  +REFP EC00068
CALL JOB:SEARCH-R1-S13D
SET P024 P006
SFTON3D P024
SMOVL C00069 BC00069 V=100.0  +MOVJ EC00069
SREFP 3 C00070 BC00070  +REFP EC00070
CALL JOB:SEARCH-R1-S13D
SET P024 P006
SFTON3D P024
SMOVL C00071 BC00071 V=100.0  +MOVJ EC00071
SFTOF3D
SMOVL C00072 BC00072 V=666.7  +MOVJ EC00072
SMOVL C00073 BC00073 V=100.0  +MOVJ EC00073
SREFP 3 C00074 BC00074  +REFP EC00074
CALL JOB:SEARCH-R1-S13D
SET P025 P006
SFTON3D P025
SMOVL C00075 BC00075 V=100.0  +MOVJ EC00075
SREFP 3 C00076 BC00076  +REFP EC00076
CALL JOB:SEARCH-R1-S13D
SET P025 P006
SFTON3D P025
SMOVL C00077 BC00077 V=100.0  +MOVJ EC00077
SFTOF3D
SMOVL C00078 BC00078 V=666.7  +MOVJ EC00078
SMOVL C00079 BC00079 V=166.7  +MOVJ EC00079
SMOVL C00080 BC00080 V=100.0  +MOVJ EC00080
SREFP 3 C00081 BC00081  +REFP EC00081
CALL JOB:SEARCH-R1-S13D
SET P026 P006
SFTON3D P026
SMOVL C00082 BC00082 V=100.0  +MOVJ EC00082
SREFP 3 C00083 BC00083  +REFP EC00083
CALL JOB:SEARCH-R1-S13D
SET P026 P006
SFTON3D P026
SMOVL C00084 BC00084 V=100.0  +MOVJ EC00084
SFTOF3D
MOVJ C00085 BC00085 VJ=100.00  +MOVJ EC00085 VJ=50.00
MOVJ C00086 BC00086 VJ=100.00  +MOVJ EC00086 VJ=50.00
MOVJ C00087 BC00087 VJ=60.00  +MOVJ EC00087 VJ=60.00
MOVJ C00088 BC00088 VJ=100.00  +MOVJ EC00088 VJ=50.00
MOVJ C00089 BC00089 VJ=60.00  +MOVJ EC00089 VJ=60.00
MOVJ C00090 BC00090 VJ=60.00  +MOVJ EC00090 VJ=60.00
SMOVL C00091 BC00091 V=166.7  +MOVJ EC00091
SREFP 3 C00092 BC00092  +REFP EC00092
CALL JOB:SEARCH-R1-S13D
SET P027 P006
SFTON3D P027
SMOVL C00093 BC00093 V=100.0  +MOVJ EC00093
SREFP 3 C00094 BC00094  +REFP EC00094
CALL JOB:SEARCH-R1-S13D
SET P027 P006
SFTON3D P027
SMOVL C00095 BC00095 V=166.7  +MOVJ EC00095
SFTOF3D
SMOVL C00096 BC00096 V=666.7  +MOVJ EC00096
SMOVL C00097 BC00097 V=100.0  +MOVJ EC00097
SREFP 3 C00098 BC00098  +REFP EC00098
CALL JOB:SEARCH-R1-S13D
SET P028 P006
SFTON3D P028
SMOVL C00099 BC00099 V=100.0  +MOVJ EC00099
SREFP 3 C00100 BC00100  +REFP EC00100
CALL JOB:SEARCH-R1-S13D
SET P028 P006
SFTON3D P028
SMOVL C00101 BC00101 V=100.0  +MOVJ EC00101
SFTOF3D
SMOVL C00102 BC00102 V=333.3  +MOVJ EC00102
SMOVL C00103 BC00103 V=100.0  +MOVJ EC00103
SREFP 3 C00104 BC00104  +REFP EC00104
CALL JOB:SEARCH-R1-S13D
SET P029 P006
SFTON3D P029
SMOVL C00105 BC00105 V=100.0  +MOVJ EC00105
SREFP 3 C00106 BC00106  +REFP EC00106
CALL JOB:SEARCH-R1-S13D
SET P029 P006
SFTON3D P029
SMOVL C00107 BC00107 V=100.0  +MOVJ EC00107
MACRO1 MJ#(0) ARGF14
'SPAWANIE 1CZ.
SMOVL C00108 BC00108 V=133.3  +MOVJ EC00108
ARCON
SMOVL C00109 BC00109 V=10.0  +MOVJ EC00109
ARCOF
SFTOF3D
SMOVL C00110 BC00110 V=250.0  +MOVJ EC00110
SMOVL C00111 BC00111 V=500.0  +MOVJ EC00111
SFTON3D P028
SMOVL C00112 BC00112 V=166.7  +MOVJ EC00112
ARCON
SMOVL C00113 BC00113 V=10.0  +MOVJ EC00113
ARCOF
SFTOF3D
SMOVL C00114 BC00114 V=166.7  +MOVJ EC00114
SMOVL C00115 BC00115 V=666.7  +MOVJ EC00115
SMOVL C00116 BC00116 V=83.3  +MOVJ EC00116
SFTON3D P027
SMOVL C00117 BC00117 V=83.3 PL=0  +MOVJ EC00117
ARCON
SMOVL C00118 BC00118 V=10.0  +MOVJ EC00118
ARCOF
SFTOF3D
SMOVL C00119 BC00119 V=166.7  +MOVJ EC00119
MOVJ C00120 BC00120 VJ=100.00  +MOVJ EC00120 VJ=50.00
MOVJ C00121 BC00121 VJ=100.00  +MOVJ EC00121 VJ=50.00
MOVJ C00122 BC00122 VJ=60.00  +MOVJ EC00122 VJ=60.00
MOVJ C00123 BC00123 VJ=100.00  +MOVJ EC00123 VJ=100.00
SFTON3D P026
SMOVL C00124 BC00124 V=133.3 PL=0  +MOVJ EC00124
ARCON
SMOVL C00125 BC00125 V=10.0  +MOVJ EC00125
ARCOF
SFTOF3D
SMOVL C00126 BC00126 V=166.7  +MOVJ EC00126
SMOVL C00127 BC00127 V=333.3  +MOVJ EC00127
SMOVL C00128 BC00128 V=166.7  +MOVJ EC00128
SFTON3D P025
SMOVL C00129 BC00129 V=166.7  +MOVJ EC00129
ARCON
SMOVL C00130 BC00130 V=10.0  +MOVJ EC00130
ARCOF
SFTOF3D
SMOVL C00131 BC00131 V=166.7  +MOVJ EC00131
SMOVL C00132 BC00132 V=166.7  +MOVJ EC00132
SFTON3D P024
SMOVL C00133 BC00133 V=166.7  +MOVJ EC00133
ARCON
SMOVL C00134 BC00134 V=10.0  +MOVJ EC00134
ARCOF
SFTOF3D
SMOVL C00135 BC00135 V=250.0  +MOVJ EC00135
SMOVL C00136 BC00136 V=416.7  +MOVJ EC00136
SFTON3D P023
SMOVL C00137 BC00137 V=166.7  +MOVJ EC00137
ARCON
SMOVL C00138 BC00138 V=10.0  +MOVJ EC00138
ARCOF
SFTOF3D
SMOVL C00139 BC00139 V=250.0  +MOVJ EC00139
SMOVL C00140 BC00140 V=500.0  +MOVJ EC00140
SFTON3D P022
SMOVL C00141 BC00141 V=166.7  +MOVJ EC00141
ARCON
SMOVL C00142 BC00142 V=10.0  +MOVJ EC00142
ARCOF
SFTOF3D
SMOVL C00143 BC00143 V=500.0  +MOVJ EC00143
SMOVL C00144 BC00144 V=500.0  +MOVJ EC00144
SFTON3D P021
SMOVL C00145 BC00145 V=133.3 PL=0  +MOVJ EC00145
ARCON
SMOVL C00146 BC00146 V=10.0  +MOVJ EC00146
ARCOF
SFTOF3D
SMOVL C00147 BC00147 V=333.3  +MOVJ EC00147
MOVJ C00148 BC00148 VJ=100.00  +MOVJ EC00148 VJ=100.00
MOVJ C00149 BC00149 VJ=100.00  +MOVJ EC00149 VJ=100.00
MOVJ C00150 BC00150 VJ=100.00  +MOVJ EC00150 VJ=100.00
SFTON3D P031
SMOVL C00151 BC00151 V=166.7  +MOVJ EC00151
ARCON
SFTON3D P030
SMOVL C00152 BC00152 V=10.0  +MOVJ EC00152
SMOVL C00153 BC00153 V=10.0  +MOVJ EC00153
ARCOF
SFTOF3D
SMOVL C00154 BC00154 V=250.0  +MOVJ EC00154
SMOVL C00155 BC00155 V=1000.0  +MOVJ EC00155
SMOVL C00156 BC00156 V=1000.0  +MOVJ EC00156
SFTON3D P032
SMOVL C00157 BC00157 V=166.7  +MOVJ EC00157
ARCON
SFTON3D P033
SMOVL C00158 BC00158 V=10.0  +MOVJ EC00158
ARCOF
SFTOF3D
SMOVL C00159 BC00159 V=500.0  +MOVJ EC00159
MOVJ C00160 BC00160 VJ=100.00  +MOVJ EC00160 VJ=30.00
MOVJ C00161 BC00161 VJ=100.00  +MOVJ EC00161 VJ=100.00
COMM MOVJ C00162 BC00162 VJ=100.00  +MOVJ EC00162 VJ=100.00
COMM MOVJ C00163 BC00163 VJ=100.00  +MOVJ EC00163 VJ=100.00
COMM MOVJ C00164 BC00164 VJ=100.00  +MOVJ EC00164 VJ=100.00
MOVJ C00165 BC00165 VJ=60.00  +MOVJ EC00165 VJ=60.00
MOVJ C00166 BC00166 VJ=60.00  +MOVJ EC00166 VJ=60.00
MOVJ C00167 BC00167 VJ=100.00  +MOVJ EC00167 VJ=100.00
MOVJ C00168 BC00168 VJ=20.00  +MOVJ EC00168 VJ=100.00
MOVJ C00169 BC00169 VJ=20.00  +MOVJ EC00169 VJ=20.00
'DRUGA POZYCJA
MOVJ C00170 BC00170 VJ=100.00  +MOVJ EC00170 VJ=100.00
MOVJ C00171 BC00171 VJ=100.00  +MOVJ EC00171 VJ=100.00
CALL JOB:CLEAN-R1_KM_NEW
MOVJ C00172 BC00172 VJ=100.00  +MOVJ EC00172 VJ=100.00
MOVJ C00173 BC00173 VJ=100.00  +MOVJ EC00173 VJ=100.00
MOVJ C00174 BC00174 VJ=100.00  +MOVJ EC00174 VJ=100.00
SMOVL C00175 BC00175 V=100.0  +MOVJ EC00175
SREFP 3 C00176 BC00176  +REFP EC00176
CALL JOB:SEARCH-R1-S13D
SET P021 P006
SFTON3D P021
SMOVL C00177 BC00177 V=100.0  +MOVJ EC00177
SREFP 3 C00178 BC00178  +REFP EC00178
CALL JOB:SEARCH-R1-S13D
SET P021 P006
SFTON3D P021
SMOVL C00179 BC00179 V=100.0  +MOVJ EC00179
SFTOF3D
SMOVL C00180 BC00180 V=333.3  +MOVJ EC00180
SMOVL C00181 BC00181 V=100.0  +MOVJ EC00181
SREFP 3 C00182 BC00182  +REFP EC00182
CALL JOB:SEARCH-R1-S13D
SET P022 P006
SFTON3D P022
SMOVL C00183 BC00183 V=100.0  +MOVJ EC00183
SREFP 3 C00184 BC00184  +REFP EC00184
CALL JOB:SEARCH-R1-S13D
SET P022 P006
SFTON3D P022
SMOVL C00185 BC00185 V=100.0  +MOVJ EC00185
SFTOF3D
SMOVL C00186 BC00186 V=333.3  +MOVJ EC00186
SMOVL C00187 BC00187 V=100.0  +MOVJ EC00187
SREFP 3 C00188 BC00188  +REFP EC00188
CALL JOB:SEARCH-R1-S13D
SET P023 P006
SFTON3D P023
SMOVL C00189 BC00189 V=100.0  +MOVJ EC00189
SREFP 3 C00190 BC00190  +REFP EC00190
CALL JOB:SEARCH-R1-S13D
SET P023 P006
SFTON3D P023
SMOVL C00191 BC00191 V=100.0  +MOVJ EC00191
SFTOF3D
SMOVL C00192 BC00192 V=333.3  +MOVJ EC00192
SMOVL C00193 BC00193 V=1000.0  +MOVJ EC00193
SMOVL C00194 BC00194 V=1000.0  +MOVJ EC00194
MOVJ C00195 BC00195 VJ=100.00  +MOVJ EC00195 VJ=100.00
MOVJ C00196 BC00196 VJ=100.00  +MOVJ EC00196 VJ=100.00
MOVJ C00197 BC00197 VJ=100.00  +MOVJ EC00197 VJ=100.00
MOVJ C00198 BC00198 VJ=100.00  +MOVJ EC00198 VJ=100.00
SMOVL C00199 BC00199 V=333.3  +MOVJ EC00199
SMOVL C00200 BC00200 V=100.0  +MOVJ EC00200
SREFP 3 C00201 BC00201  +REFP EC00201
CALL JOB:SEARCH-R1-S13D
SET P024 P006
SFTON3D P024
SMOVL C00202 BC00202 V=100.0  +MOVJ EC00202
SREFP 3 C00203 BC00203  +REFP EC00203
CALL JOB:SEARCH-R1-S13D
SET P024 P006
SFTON3D P024
SMOVL C00204 BC00204 V=100.0  +MOVJ EC00204
SFTOF3D
SMOVL C00205 BC00205 V=333.3  +MOVJ EC00205
SMOVL C00206 BC00206 V=100.0  +MOVJ EC00206
SREFP 3 C00207 BC00207  +REFP EC00207
CALL JOB:SEARCH-R1-S13D
SET P025 P006
SFTON3D P025
SMOVL C00208 BC00208 V=100.0  +MOVJ EC00208
SREFP 3 C00209 BC00209  +REFP EC00209
CALL JOB:SEARCH-R1-S13D
SET P025 P006
SFTON3D P025
SMOVL C00210 BC00210 V=100.0  +MOVJ EC00210
SFTOF3D
SMOVL C00211 BC00211 V=500.0  +MOVJ EC00211
SMOVL C00212 BC00212 V=100.0  +MOVJ EC00212
SREFP 3 C00213 BC00213  +REFP EC00213
CALL JOB:SEARCH-R1-S13D
SET P026 P006
SFTON3D P026
SMOVL C00214 BC00214 V=60.0  +MOVJ EC00214
SREFP 3 C00215 BC00215  +REFP EC00215
CALL JOB:SEARCH-R1-S13D
SET P026 P006
SFTON3D P026
SMOVL C00216 BC00216 V=60.0  +MOVJ EC00216
SFTOF3D
MOVJ C00217 BC00217 VJ=100.00  +MOVJ EC00217 VJ=50.00
MOVJ C00218 BC00218 VJ=100.00  +MOVJ EC00218 VJ=50.00
SMOVL C00219 BC00219 V=100.0  +MOVJ EC00219
SREFP 3 C00220 BC00220  +REFP EC00220
CALL JOB:SEARCH-R1-S13D
SET P027 P006
SFTON3D P027
SMOVL C00221 BC00221 V=100.0  +MOVJ EC00221
SREFP 3 C00222 BC00222  +REFP EC00222
CALL JOB:SEARCH-R1-S13D
SET P027 P006
SFTON3D P027
SMOVL C00223 BC00223 V=100.0  +MOVJ EC00223
SFTOF3D
SMOVL C00224 BC00224 V=250.0  +MOVJ EC00224
SMOVL C00225 BC00225 V=100.0  +MOVJ EC00225
SREFP 3 C00226 BC00226  +REFP EC00226
CALL JOB:SEARCH-R1-S13D
SET P028 P006
SFTON3D P028
SMOVL C00227 BC00227 V=100.0  +MOVJ EC00227
SREFP 3 C00228 BC00228  +REFP EC00228
CALL JOB:SEARCH-R1-S13D
SET P028 P006
SFTON3D P028
SMOVL C00229 BC00229 V=100.0  +MOVJ EC00229
SFTOF3D
SMOVL C00230 BC00230 V=416.7  +MOVJ EC00230
SMOVL C00231 BC00231 V=10.0  +MOVJ EC00231
SREFP 3 C00232 BC00232  +REFP EC00232
CALL JOB:SEARCH-R1-S13D
SET P029 P006
SFTON3D P029
SMOVL C00233 BC00233 V=100.0  +MOVJ EC00233
SREFP 3 C00234 BC00234  +REFP EC00234
CALL JOB:SEARCH-R1-S13D
SET P029 P006
SFTON3D P029
SMOVL C00235 BC00235 V=100.0  +MOVJ EC00235
MOVJ C00236 BC00236 VJ=100.00  +MOVJ EC00236 VJ=100.00
MOVJ C00237 BC00237 VJ=100.00  +MOVJ EC00237 VJ=100.00
MOVJ C00238 BC00238 VJ=100.00  +MOVJ EC00238 VJ=100.00
SMOVL C00239 BC00239 V=10.0  +MOVJ EC00239
SREFP 3 C00240 BC00240  +REFP EC00240
CALL JOB:SEARCH-R1-S13D
SET P030 P006
SFTON3D P030
SMOVL C00241 BC00241 V=100.0  +MOVJ EC00241
SREFP 3 C00242 BC00242  +REFP EC00242
CALL JOB:SEARCH-R1-S13D
SET P030 P006
SFTON3D P030
SMOVL C00243 BC00243 V=100.0  +MOVJ EC00243
SFTOF3D
SMOVL C00244 BC00244 V=416.7  +MOVJ EC00244
SMOVL C00245 BC00245 V=100.0  +MOVJ EC00245
SREFP 3 C00246 BC00246  +REFP EC00246
CALL JOB:SEARCH-R1-S13D
SET P031 P006
SFTON3D P031
SMOVL C00247 BC00247 V=100.0  +MOVJ EC00247
SREFP 3 C00248 BC00248  +REFP EC00248
CALL JOB:SEARCH-R1-S13D
SET P031 P006
SFTON3D P031
SMOVL C00249 BC00249 V=100.0  +MOVJ EC00249
SFTOF3D
SMOVL C00250 BC00250 V=500.0  +MOVJ EC00250
SMOVL C00251 BC00251 V=1000.0  +MOVJ EC00251
SMOVL C00252 BC00252 V=500.0  +MOVJ EC00252
SMOVL C00253 BC00253 V=100.0  +MOVJ EC00253
SREFP 3 C00254 BC00254  +REFP EC00254
CALL JOB:SEARCH-R1-S13D
SET P033 P006
SFTON3D P033
SMOVL C00255 BC00255 V=100.0  +MOVJ EC00255
SREFP 3 C00256 BC00256  +REFP EC00256
CALL JOB:SEARCH-R1-S13D
SET P033 P006
SFTON3D P033
SMOVL C00257 BC00257 V=100.0  +MOVJ EC00257
SFTOF3D
SMOVL C00258 BC00258 V=416.7  +MOVJ EC00258
SMOVL C00259 BC00259 V=100.0  +MOVJ EC00259
SREFP 3 C00260 BC00260  +REFP EC00260
CALL JOB:SEARCH-R1-S13D
SET P032 P006
SFTON3D P032
SMOVL C00261 BC00261 V=100.0  +MOVJ EC00261
SREFP 3 C00262 BC00262  +REFP EC00262
CALL JOB:SEARCH-R1-S13D
SET P032 P006
SFTON3D P032
SMOVL C00263 BC00263 V=100.0  +MOVJ EC00263
MACRO1 MJ#(0) ARGF14
SMOVL C00264 BC00264 V=166.7  +MOVJ EC00264
ARCON
SFTON3D P033
SMOVL C00265 BC00265 V=9.2  +MOVJ EC00265
ARCOF
SFTOF3D
SMOVL C00266 BC00266 V=416.7  +MOVJ EC00266
SMOVL C00267 BC00267 V=1000.0  +MOVJ EC00267
SMOVL C00268 BC00268 V=416.7  +MOVJ EC00268
SFTON3D P030
SMOVL C00269 BC00269 V=133.3  +MOVJ EC00269
ARCON
SFTON3D P031
SMOVL C00270 BC00270 V=8.3  +MOVJ EC00270
ARCOF
SFTOF3D
SMOVL C00271 BC00271 V=416.7  +MOVJ EC00271
MOVJ C00272 BC00272 VJ=100.00  +MOVJ EC00272 VJ=100.00
MOVJ C00273 BC00273 VJ=100.00  +MOVJ EC00273 VJ=100.00
MOVJ C00274 BC00274 VJ=100.00  +MOVJ EC00274 VJ=100.00
'BRAK POM SPR CZY OK
SFTON3D P029
SMOVL C00275 BC00275 V=133.3  +MOVJ EC00275
ARCON
MOVL C00276 BC00276 V=10.0  +MOVJ EC00276 VJ=15.00
ARCOF
SFTOF3D
MOVJ C00277 BC00277 VJ=100.00  +MOVJ EC00277 VJ=15.00
SFTON3D P028
SMOVL C00278 BC00278 V=133.3  +MOVJ EC00278
ARCON
SMOVL C00279 BC00279 V=10.0  +MOVJ EC00279
ARCOF
SFTOF3D
SMOVL C00280 BC00280 V=500.0  +MOVJ EC00280
SMOVL C00281 BC00281 V=833.3  +MOVJ EC00281
SFTON3D P027
SMOVL C00282 BC00282 V=133.3  +MOVJ EC00282
ARCON
SMOVL C00283 BC00283 V=10.0  +MOVJ EC00283
ARCOF
SFTOF3D
SMOVL C00284 BC00284 V=250.0  +MOVJ EC00284
SMOVL C00285 BC00285 V=500.0  +MOVJ EC00285
SMOVL C00286 BC00286 V=333.3  +MOVJ EC00286
SFTON3D P026
SMOVL C00287 BC00287 V=133.3  +MOVJ EC00287
ARCON
SMOVL C00288 BC00288 V=10.0  +MOVJ EC00288
ARCOF
SFTOF3D
SMOVL C00289 BC00289 V=250.0  +MOVJ EC00289
SFTON3D P025
SMOVL C00290 BC00290 V=250.0  +MOVJ EC00290
SMOVL C00291 BC00291 V=133.3  +MOVJ EC00291
ARCON
SMOVL C00292 BC00292 V=10.0  +MOVJ EC00292
ARCOF
SFTOF3D
SMOVL C00293 BC00293 V=250.0  +MOVJ EC00293
SMOVL C00294 BC00294 V=500.0  +MOVJ EC00294
SFTON3D P024
SMOVL C00295 BC00295 V=133.3  +MOVJ EC00295
ARCON
SMOVL C00296 BC00296 V=10.0  +MOVJ EC00296
ARCOF
SMOVL C00297 BC00297 V=666.7  +MOVJ EC00297
SMOVL C00298 BC00298 V=1000.0  +MOVJ EC00298
SMOVL C00299 BC00299 V=333.3  +MOVJ EC00299
SMOVL C00300 BC00300 V=1000.0  +MOVJ EC00300
SMOVL C00301 BC00301 V=1000.0  +MOVJ EC00301
SMOVL C00302 BC00302 V=1000.0  +MOVJ EC00302
SMOVL C00303 BC00303 V=666.7  +MOVJ EC00303
SFTON3D P021
SMOVL C00304 BC00304 V=133.3  +MOVJ EC00304
ARCON
SMOVL C00305 BC00305 V=10.0  +MOVJ EC00305
ARCOF
SFTOF3D
SMOVL C00306 BC00306 V=166.7  +MOVJ EC00306
SMOVL C00307 BC00307 V=666.7  +MOVJ EC00307
SFTON3D P022
SMOVL C00308 BC00308 V=133.3  +MOVJ EC00308
ARCON
SMOVL C00309 BC00309 V=10.0  +MOVJ EC00309
ARCOF
SFTOF3D
SMOVL C00310 BC00310 V=133.3  +MOVJ EC00310
SMOVL C00311 BC00311 V=666.7  +MOVJ EC00311
SFTON3D P023
SMOVL C00312 BC00312 V=133.3  +MOVJ EC00312
ARCON
SMOVL C00313 BC00313 V=10.0  +MOVJ EC00313
ARCOF
SFTOF3D
SMOVL C00314 BC00314 V=666.7  +MOVJ EC00314
MOVJ C00315 BC00315 VJ=100.00  +MOVJ EC00315 VJ=100.00
MOVJ C00316 BC00316 VJ=100.00  +MOVJ EC00316 VJ=100.00
END
